Fanuc KAREL source: kt00544.KL

-- PROVISIONAL review KL for V1013-1; original PC SHA256 2b7d58b27e10d1096e20ee84cabe041aa2778272dfda308be053227b4fc61135
-- Incomplete behavior may be omitted. Consult companion uncertainty JSON. Do not deploy.
PROGRAM KT00544
%NOLOCKGROUP
-- UNRESOLVED_DECL P1 type=000199
-- UNRESOLVED_DECL P2 type=000106
-- UNRESOLVED_DECL OUT type=000101
BEGIN
  -- UNRESOLVED_PC offsets 5-20; opcodes 2E,22,32,35
  -- UNRESOLVED_PC offsets 25-59; opcodes 49,7E,49,7E,60,4A
  -- UNRESOLVED_PC offsets 64-68; opcodes 7F
END KT00544
